// TIA Portal V17 export
// export: Created 2024-09-02T12:49:59.0332071Z, ExportSetting WithDefaults, DisplayName Totally Integrated Automation Portal, DisplayVersion V17, DisplayName TIA Portal Openness, DisplayVersion V17, DisplayName TIA Portal Version Control Interface, DisplayVersion V17, DisplayName STEP 7 Professional, DisplayVersion V17, DisplayName STEP 7 Safety, DisplayVersion V17, DisplayName WinCC Professional, DisplayVersion V17
DATA_BLOCK "LTLL_Config"   // DB555
TITLE = LTLL_Config
{ DB_Accessible_From_OPC_UA := 'FALSE' }
AUTHOR : Siemens
FAMILY : HMI_Lite
NAME : LTLL_Config
VERSION : 8.10
// stored: AutoNumber true, DBAccessibleFromOPCUA false, IsOnlyStoredInLoadMemory false, IsWriteProtectedInAS false
   STRUCT
      LTLL_Config : Array[0..1] of "LTLL_typeConfig";
   END_STRUCT;
BEGIN
   LTLL_Config[0..1]."version".high := 16#08;
   LTLL_Config[0..1]."version".middle := 16#01;
   LTLL_Config[0..1]."version".low := 16#00;
   LTLL_Config[0].licensing.licenseNumber := 'N6OV08904';
   LTLL_Config[0].licensing.licenseKey[0] := 16#21;
   LTLL_Config[0].licensing.licenseKey[1] := 16#51;
   LTLL_Config[0].licensing.licenseKey[2] := 16#A0;
   LTLL_Config[0].licensing.licenseKey[3] := 16#EA;
   LTLL_Config[0].licensing.licenseKey[4] := 16#C0;
   LTLL_Config[0].licensing.licenseKey[5] := 16#12;
   LTLL_Config[0].licensing.licenseKey[6] := 16#F8;
   LTLL_Config[0].licensing.licenseKey[7] := 16#C0;
   LTLL_Config[0].licensing.licenseKey[8] := 16#70;
   LTLL_Config[0].licensing.licenseKey[9] := 16#F4;
   LTLL_Config[0].header.useTextLayout := True;
   LTLL_Config[0].screenCounter.TimeValueHideReset := T#5s;
END_DATA_BLOCK
